// TIA Portal V18 export
DATA_BLOCK "Scanner1LoadData"   // DB530
{ S7_Optimized_Access := 'FALSE' }
// stored: AutoNumber false
   VAR
      "PLC.Station1DMXCode" : Int;
      "PLC.Station1RecipeNo" : Int;
      "PLC.PartTypeID" : String[128];
      Spare : Byte;
      "MES.ErrorCode" : Int;
      "MES.StatusBits" : DInt;
      "MES.Cycle_ID" : DInt;
      "MES.Unit_ParttypeID" : Int;
   END_VAR
BEGIN
END_DATA_BLOCK
